(* PLC project execute-test.project, CODESYS CODESYS V3.5 SP22 Patch 1 *)
(* stored: creationDateTime 2026-08-28T09:52:30.8266995, modificationDateTime 2026-08-28T09:52:13.9833565 *)

PROGRAM PLC_PRG
  VAR
    myValue : INT;
    myNewValue : INT;
    myContact : BOOL;
    myCoil : BOOL;
    myValue_1 : INT;
    myNewValue_1 : INT;
    myContact_1 : BOOL;
    myCoil_1 : BOOL;
  END_VAR

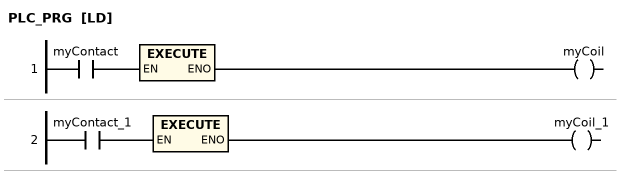
(* LD diagram, written out as Structured Text *)
(* ST Block Comment *)
(* --- network: ST Block Network --- *)
IF myContact THEN
  // escaping test: < > <= >= <>
  (* block comment: ampersand & , less-than < , greater-than > , quotes 'single' "double" *)
  IF myValue < 10 AND myContact THEN
      myNewValue := myValue + 1;
  ELSIF (myValue >= 10) AND (myValue <= 100) THEN
      myNewValue := myValue - 1;
  ELSIF myValue <> 0 THEN
      myNewValue := 0;
  ELSE
      myNewValue := -1;
  END_IF;
  
  FOR myValue := 0 TO 5 BY 1 DO
      myNewValue := myNewValue + myValue;
  END_FOR;
  
  CASE myNewValue OF
      0, 1: myCoil := TRUE;
      2..5: myCoil := FALSE;
  ELSE
      myCoil := myContact;
  END_CASE;
END_IF;
myCoil := myContact;
(* ST Block Comment 1 *)
(* --- network: ST Block Network 1 --- *)
IF myContact_1 THEN
  // Comment in ST Block 1
  myNewValue_1 := myValue_1 + 111;
END_IF;
myCoil_1 := myContact_1;
END_PROGRAM

PROGRAM FBD_Test_Execute
  VAR
    myNewVarFBD : INT;
  END_VAR

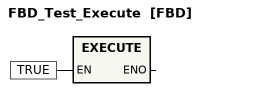
(* FBD diagram, written out as Structured Text *)
IF TRUE THEN
  // FBD escaping test: a < b , c > d , e <> f
  IF myNewVarFBD < 100 AND myNewVarFBD <> 0 THEN
      myNewVarFBD := myNewVarFBD + 1;
  ELSE
      myNewVarFBD := 0;
  END_IF;
END_IF;
END_PROGRAM
